# EPICS autosave request: ipApp/Db/BK9130_settings.req
# FILE... BK9130_settings.req
$(P)BK9130:$(PS):CH1_Vset
$(P)BK9130:$(PS):CH1_Iset
$(P)BK9130:$(PS):CH2_Vset
$(P)BK9130:$(PS):CH2_Iset
$(P)BK9130:$(PS):CH3_Vset
$(P)BK9130:$(PS):CH3_Iset
$(P)BK9130:$(PS):get_Vmeas.SCAN
